{attribute 'reflection'}
FUNCTION_BLOCK TNamedBase
VAR
	{attribute 'instance-path'}
    {attribute 'no_init'}
	name : STRING;
	_instanceName : STRING; // name minus project name etc.
	_instanceSet : BOOL;
END_VAR

PROPERTY FINAL InstanceName : T_MaxString;
GET
IF NOT _instanceSet THEN
	setInstanceName();
END_IF

InstanceName := _instanceName;
END_GET
END_PROPERTY

METHOD LogError
VAR_INPUT
	Msg : T_MaxString;
END_VAR
F_LogError(
	F_Concat3(InstanceName , ': ', Msg)
);
END_METHOD

METHOD LogInfo
VAR_INPUT
	Msg : T_MaxString;
END_VAR
F_LogInfo(
	F_Concat3(InstanceName , ': ', Msg)
);
END_METHOD

METHOD LogWarning
VAR_INPUT
	Msg : T_MaxString;
END_VAR
F_LogWarning(
	F_Concat3(InstanceName , ': ', Msg)
);
END_METHOD

METHOD PRIVATE setInstanceName 
VAR
	charsToDeleteFromPath : INT;
END_VAR
// format is  Solution_Name.ProjectName.FirstDeclaredPOU.etc.etc... 

//Remove Solution_Name
charsToDeleteFromPath := FIND( name, '.' );
_instanceName := DELETE( name, charsToDeleteFromPath, 1 );

//Remove ProjectName
charsToDeleteFromPath := FIND( _instanceName, '.' );

//gives us just "FirstDeclaredPOU.etc.etc..." from above.
_instanceName := DELETE( _instanceName, charsToDeleteFromPath, 1 );

_instanceSet := TRUE;
END_METHOD

END_FUNCTION_BLOCK

(* stored: Version 1.1.0.1, ProductVersion 3.1.4022.10
   POU TNamedBase: Id {747db62b-b007-4b65-974e-3e30c9f6f818}, SpecialFunc None
   Property InstanceName: Id {b025274c-dbbe-41b4-9d4a-6b264880646b}
   Get Get: Id {c76f2db8-929e-42c3-879d-8eaff2d7bbd0}
   Method LogError: Id {68460783-e2b1-4495-92bf-87f826bbe299}
   Method LogInfo: Id {d072dd6f-6f37-41d6-8089-6cac6bd97a28}
   Method LogWarning: Id {6676ad4f-087f-4dd6-bf57-0b34c5abe60e}
   Method setInstanceName: Id {d237b876-4874-4101-9aea-59f0ea3e9132} *)
